PROGRAM P_InfluxDatabaseWriter
VAR
	Data : REFERENCE TO FB_InfluxDataCollector := P_InfluxDataCollector.InfluxData; 	

	Sender : FB_InfluxDataSender; 
	
	WriteSucces : BOOL; 
END_VAR

(* This Sender Program Should be run at 10ms ScanTime in seperate task (can be same CPU) from DataCollector *)

IF Main.EmulatedState = E_EmulatedState.PhysicalPlant THEN
	Sender(	Data				:= Data,
			Ip					:= '10.10.0.122',
			Port				:= 8086,
			GlobalWriteSucces 	=> WriteSucces); 
ELSIF Main.EmulatedState = E_EmulatedState.VirtualPlant THEN
	Sender(	Data				:= Data,
			Ip					:= '127.0.0.1',
			Port				:= 8086,
			GlobalWriteSucces 	=> WriteSucces); 	

END_IF



// =============== Read Values from Influxdb

END_PROGRAM

(* stored: Version 1.1.0.1, ProductVersion 3.1.4022.11
   POU P_InfluxDatabaseWriter: Id {51cfc44b-9173-4a49-8914-2b4985a65a2e}, SpecialFunc None *)
